(* IEC 61131-3 sources: LogicFuzz/ExampleTestProgram/codesysLogicInstruction, 3 files *)

(* ---- sysmemcpy.st ---- *)
PROGRAM PLC_PRG
VAR
    Dest : DINT;
    Src : DINT;
    udiCount : DINT;
END_VAR

Dest := 12345678;
Src := 87654321;
udiCount := 4;

SysMemCpy( Dest,Src,udiCount);

(* ---- sysmemmove.st ---- *)
PROGRAM PLC_PRG
VAR
    Dest : DINT;
    Src : DINT;
    udiCount : DINT;
END_VAR

Dest := 12345678;
Src := 87654321;
udiCount := 4;

SysMemMove( Dest, Src, udiCount );

(* ---- syssockconnect.st ---- *)
PROGRAM PLC_PRG
VAR_INPUT
diSocket: DINT;
pSockAddr: DWORD;
diSockAddrSize: DINT;
END_VAR

diSocket := 1;
pSockAddr := 2;
diSockAddrSize := 3;
//Execute the SysSockConnect instruction
SysSockConnect(diSocket,
pSockAddr, diSockAddrSize);
